FUNCTION_BLOCK FB_ClampJog
VAR_INPUT
	Rst	:BOOL;
END_VAR
VAR_OUTPUT
END_VAR
VAR
	iClampDn1,iClampUp1	:INT;
	rtClampDn	:R_TRIG;
	rtClampUp	:R_TRIG;
	flag00,flag01: BOOL;
	tonPedalClampDn	:TON;
	tonPedalClampUp	:TON;
	flag02: BOOL;
	bUnClamp: BOOL;
	bClamp: BOOL;
END_VAR

IF Rst THEN
	iClampDn1	:=30;	iClampUp1	:=2;
END_IF

flag00:=stFolder.Status.Slitter_AtHome AND stFolder.Status.ApronTopFold_AtHome AND stFolder.Status.ApronBtmFold_AtHome;
bUnClamp:= pedal_UnClamp;
bClamp	:= pedal_Clamp;

flag01:=flag00 AND stFolder.Status.Table_AtHome;
tonPedalClampDn(IN:=bClamp AND NOT bUnClamp , PT:=T#500MS , Q=> , ET=> );
tonPedalClampUp(IN:=NOT bClamp AND bUnClamp , PT:=T#500MS , Q=> , ET=> );
rtClampDn(CLK:=tonPedalClampDn.Q , Q=> );
rtClampUp(CLK:=tonPedalClampUp.Q , Q=> );


//flag00:=TRUE;
//flag01:=TRUE;
CASE iClampDn1 OF
	0:
		IF rtClampDn.Q AND flag01 THEN
			IF NOT stFolder.Status.Clamp_LtHalfPoint THEN
				iClampDn1	:=10;
			ELSIF stFolder.Status.Clamp_LtHalfPoint THEN
				iClampDn1	:=20;
			ELSE
				iClampDn1	:=30;
			END_IF
		END_IF
	10:
		Out_ClampDown	:=TRUE;
		Out_ClampUp		:=FALSE;
		iClampDn1	:=SEL(NOT bClamp OR stFolder.Status.Clamp_LtHalfPoint,10,30);
	20:
		Out_ClampDown	:=TRUE;
		Out_ClampUp		:=FALSE;
		//flag01	:= (stFolder.Status.Clamp_AtZeroPoint AND stFolder.Status.Clamp_AtPressPoint);
		//flag01	:= (stFolder.Status.Clamp_AtZeroPoint);
		iClampDn1	:=SEL((NOT bClamp OR flag02),20,30);
	30:
		Out_ClampDown:= Out_ClampUp :=FALSE;
		iClampDn1	:=0;
END_CASE

CASE iClampUp1 OF
	0: 
		IF flag00 AND rtClampUp.Q THEN
			iClampUp1	:=1;
			iClampDn1	:=0;
		END_IF
		
	1:
		Out_ClampUp		:=TRUE;
		Out_ClampDown	:=FALSE;
		iClampUp1	:=SEL(NOT bUnClamp OR stFolder.ClampHt_ActPos>=stFolderPara.Clamp_MaxPos,1,2);
//		iClampUp1	:=SEL(NOT bUnClamp ,1,2);
	2:
		Out_ClampUp	:= Out_ClampDown	:=FALSE;
		iClampUp1	:=0;
		
		
END_CASE

END_FUNCTION_BLOCK

(* stored: Version 1.1.0.1, ProductVersion 3.1.4024.15
   POU FB_ClampJog: Id {de6e07fb-f5e8-49ac-896a-08339a2d3ce1}, SpecialFunc None *)
